// TIA Portal V17 export
FUNCTION "FC_MainControl" : Void   // FC, LAD
{ S7_Optimized_Access := 'TRUE' }
   VAR_TEMP
      风机控制输出值 : Real;
      风压过渡 : Int;
   END_VAR
BEGIN

REGION Network 1: 风机输出
   // 风机运行条件判断：运行按接通且无故障反馈时驱动风机运行线圈。自动/手动模式选择：手动OFF时MOVE自动输出值，手动ON时MUL手动频率乘2.0，二者互斥写入风机控制输出。
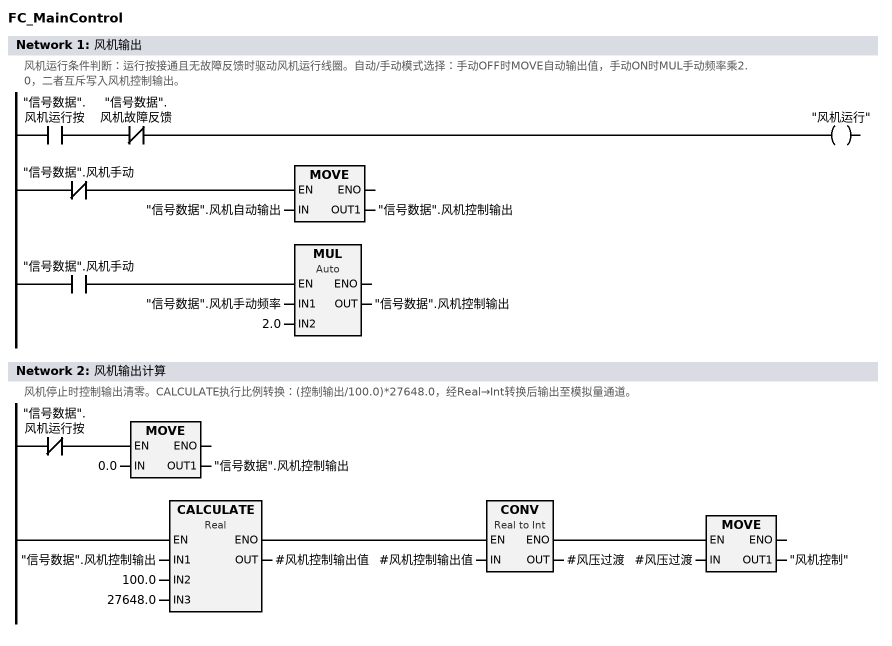
   RUNG wire#powerrail
      Contact( "信号数据".风机运行按 )
      I_Contact( "信号数据".风机故障反馈 )
      Coil( "风机运行" )
   END_RUNG
   RUNG wire#powerrail
      I_Contact( "信号数据".风机手动 )
      { S7_GenerateENO := "TRUE" } Move(in := "信号数据".风机自动输出, out1 => "信号数据".风机控制输出)
   END_RUNG
   RUNG wire#powerrail
      Contact( "信号数据".风机手动 )
      { S7_GenerateENO := "TRUE" } Mul(in1 := "信号数据".风机手动频率, in2 := 2.0, out => "信号数据".风机控制输出)
   END_RUNG
   // the same network as SCL:
   "风机运行" := "信号数据".风机运行按 AND NOT "信号数据".风机故障反馈;
   IF NOT "信号数据".风机手动 THEN "信号数据".风机控制输出 := "信号数据".风机自动输出; END_IF;
   IF "信号数据".风机手动 THEN "信号数据".风机控制输出 := "信号数据".风机手动频率 * 2.0; END_IF;
END_REGION

REGION Network 2: 风机输出计算
   // 风机停止时控制输出清零。CALCULATE执行比例转换：(控制输出/100.0)*27648.0，经Real→Int转换后输出至模拟量通道。
   RUNG wire#powerrail
      I_Contact( "信号数据".风机运行按 )
      { S7_GenerateENO := "TRUE" } Move(in := 0.0, out1 => "信号数据".风机控制输出)
   END_RUNG
   RUNG wire#powerrail
      { S7_Templates := "SrcType := Real"; S7_GenerateENO := "TRUE"; S7_Expression := "(IN1/IN2)*IN3" } Calculate(in1 := "信号数据".风机控制输出, in2 := 100.0, in3 := 27648.0, out => #风机控制输出值)
      { S7_Templates := "[SrcType := Real, DestType := Int]" } Convert(in := #风机控制输出值, out => #风压过渡)
      { S7_GenerateENO := "TRUE" } Move(in := #风压过渡, out1 => "风机控制")
   END_RUNG
   // the same network as SCL:
   // ENO of a box is taken as its EN; it also drops when the box reports an error
   IF NOT "信号数据".风机运行按 THEN "信号数据".风机控制输出 := 0.0; END_IF;
   #风机控制输出值 := ("信号数据".风机控制输出/100.0)*27648.0;
   #风压过渡 := REAL_TO_INT(#风机控制输出值);
   "风机控制" := #风压过渡;
END_REGION
END_FUNCTION
